(* CoDeSys 2.3 export: F_READ_TACK_VALVE_CFG.EXP *)

(* POU FUN/PARAMETERS/F_READ_TACK_VALVE_CFG, ST *)
FUNCTION F_READ_TACK_VALVE_CFG : BOOL
VAR_INPUT
	sHead : STRING;
	rTime : REAL;
END_VAR
VAR_IN_OUT
	stConfig : ST_TACK_VALVE_CFG;
	fbIdList : FB_IDLIST;
END_VAR
VAR
END_VAR
stConfig.Cycle    := rTime;
stConfig.TimeMax  := F_IDLIST_GETREAL( CONCAT(sHead, '_TimeMax'   ), fbIdList );

stConfig.Hyst_HeelH := F_IDLIST_GETREAL( CONCAT(sHead, '_Hyst_HeelH' ), fbIdList );
stConfig.Hyst_HeelL := F_IDLIST_GETREAL( CONCAT(sHead, '_Hyst_HeelL' ), fbIdList );
stConfig.Hyst_Time  := F_IDLIST_GETREAL( CONCAT(sHead, '_Hyst_Time'  ), fbIdList );
END_FUNCTION
